# EPICS substitutions: scllrfApp/Db/PRCRegisters.substitutions
file scllrfPRC.template
{
	{ NULL = NULL }
}

file scllrfCommon.template
{
	{ NULL = NULL }
}
